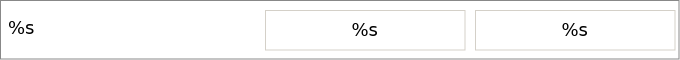
VISUALIZATION SingleRecipesParameterTypeString  // 680x60
VAR_IN_OUT
	stRecipeParameter : ST_VisuCtrlRecipeParameter;
END_VAR
    Textfield (265,10 200x40), "%s", text variable: stRecipeParameter.sValue
        OnMouseClick: write the text variable via VisuDialogs.Keypad
    Textfield (475,10 200x40), "%s", text variable: stRecipeParameter.sFileValue
    Textfield (5,8 250x40), "%s", text variable: stRecipeParameter.sName
END_VISUALIZATION

(* stored: Version 1.1.0.1, ProductVersion 3.1.4024.9
   Visu SingleRecipesParameterTypeString: Id {0787835b-8aec-48f6-ba63-f6fe4fb2379f} *)
